{attribute 'GeneratedUsingTerminal: EP2809-0042-0018'}
{attribute addProperty BoxType "EP2809-0042-0018"}
{attribute addProperty Id "DO_X01_4AT %Q*DO_X_42CA91F71DO_X01_2AT %Q*DO_X_42CA91F71DO_X02_4AT %Q*DO_X_42CA91F71DO_X02_2AT %Q*DO_X_42CA91F71DO_X03_4AT %Q*DO_X_42CA91F71DO_X03_2AT %Q*DO_X_42CA91F71DO_X04_4AT %Q*DO_X_42CA91F71DO_X04_2AT %Q*DO_X_42CA91F71DO_X05_4AT %Q*DO_X_42CA91F71DO_X05_2AT %Q*DO_X_42CA91F71DO_X06_4AT %Q*DO_X_42CA91F71DO_X06_2AT %Q*DO_X_42CA91F71DO_X07_4AT %Q*DO_X_42CA91F71DO_X07_2AT %Q*DO_X_42CA91F71DO_X08_4AT %Q*DO_X_42CA91F71DO_X08_2AT %Q*DO_X_42CA91F71WcStateAT %I*WcState_0B2B16F91InfoDataAT %I*InfoData_6F19DB2B2"}
{attribute addProperty CRC "593641116"}
{attribute addProperty Size "19"}
TYPE EP2809_23623E9C EXTENDS EtcSlaveTerminalBase_947E5A46 :
STRUCT
	{attribute addProperty Name "DO_X01_4"}
	DO_X01_4 : DO_X_42CA91F7;
	{attribute addProperty Name "DO_X01_2"}
	DO_X01_2 : DO_X_42CA91F7;
	{attribute addProperty Name "DO_X02_4"}
	DO_X02_4 : DO_X_42CA91F7;
	{attribute addProperty Name "DO_X02_2"}
	DO_X02_2 : DO_X_42CA91F7;
	{attribute addProperty Name "DO_X03_4"}
	DO_X03_4 : DO_X_42CA91F7;
	{attribute addProperty Name "DO_X03_2"}
	DO_X03_2 : DO_X_42CA91F7;
	{attribute addProperty Name "DO_X04_4"}
	DO_X04_4 : DO_X_42CA91F7;
	{attribute addProperty Name "DO_X04_2"}
	DO_X04_2 : DO_X_42CA91F7;
	{attribute addProperty Name "DO_X05_4"}
	DO_X05_4 : DO_X_42CA91F7;
	{attribute addProperty Name "DO_X05_2"}
	DO_X05_2 : DO_X_42CA91F7;
	{attribute addProperty Name "DO_X06_4"}
	DO_X06_4 : DO_X_42CA91F7;
	{attribute addProperty Name "DO_X06_2"}
	DO_X06_2 : DO_X_42CA91F7;
	{attribute addProperty Name "DO_X07_4"}
	DO_X07_4 : DO_X_42CA91F7;
	{attribute addProperty Name "DO_X07_2"}
	DO_X07_2 : DO_X_42CA91F7;
	{attribute addProperty Name "DO_X08_4"}
	DO_X08_4 : DO_X_42CA91F7;
	{attribute addProperty Name "DO_X08_2"}
	DO_X08_2 : DO_X_42CA91F7;
	{attribute addProperty Name "WcState"}
	WcState : WcState_0B2B16F9;
	{attribute addProperty Name "InfoData"}
	InfoData : InfoData_6F19DB2B;
END_STRUCT
END_TYPE

(* stored: Version 1.2.0.0, ProductVersion 3.1.4024.9
   DUT EP2809_23623E9C: Id {1618ec0a-3e0a-4210-81d4-e1f3f67ff6ee} *)
